FUNCTION_BLOCK GR_CMD (* Basic Function Block Type *)
  (* Standard: 61499-2 *)
  (* Version 0.0, 18/07/2022, Etienne, Schneider Electric, Template *)
  PACKAGE Main;
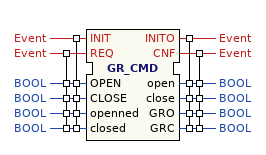
  EVENT_INPUT
    INIT WITH OPEN, CLOSE, openned, closed; (* Initialization Request *)
    REQ WITH OPEN, CLOSE, openned, closed; (* Normal Execution Request *)
  END_EVENT
  EVENT_OUTPUT
    INITO WITH open, close, GRO, GRC; (* Initialization Confirm *)
    CNF WITH open, close, GRO, GRC; (* Execution Confirmation *)
  END_EVENT
  VAR_INPUT
    OPEN : BOOL;
    CLOSE : BOOL;
    openned : BOOL;
    closed : BOOL;
  END_VAR
  VAR_OUTPUT
    open : BOOL;
    close : BOOL;
    GRO : BOOL;
    GRC : BOOL;
  END_VAR
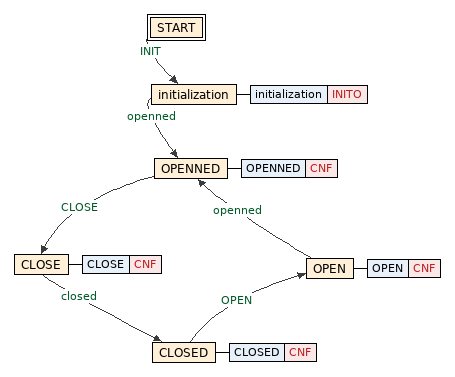
  EC_STATES
    START; (* Initial State *)
    initialization : initialization -> INITO;
    OPEN : OPEN -> CNF;
    CLOSE : CLOSE -> CNF;
    OPENNED : OPENNED -> CNF;
    CLOSED : CLOSED -> CNF;
  END_STATES
  EC_TRANSITIONS
    initialization TO OPENNED := openned;
    OPEN TO OPENNED := openned;
    CLOSE TO CLOSED := closed;
    OPENNED TO CLOSE := CLOSE;
    CLOSED TO OPEN := OPEN;
    START TO initialization := INIT;
  END_TRANSITIONS
  ALGORITHM initialization IN ST:
;
open:=TRUE;
close:=FALSE;
  END_ALGORITHM
  ALGORITHM OPEN IN ST:
open:=TRUE;
close:=FALSE;
  END_ALGORITHM
  ALGORITHM CLOSE IN ST:
open:=FALSE;
close:=TRUE;
  END_ALGORITHM
  ALGORITHM OPENNED IN ST:
GRO:=TRUE;
GRC:=FALSE;
  END_ALGORITHM
  ALGORITHM CLOSED IN ST:
GRO:=FALSE;
GRC:=TRUE;
  END_ALGORITHM
END_FUNCTION_BLOCK
